PROGRAM Note
VAR
END_VAR

進料台車:
	編碼器對應實際距離: 0.025mm/p
	歸零偏移 : 22mm  > 880p
	最大行程 編碼器 108466 p 實際 2710 mm
	進料範圍 0 - 1000
	暫存範圍 1300 - 2800
	
	30HZ = 164mm/S
	 3HZ =  16mm/S
	 
進料流程:
1.將進料區的工件全部往定位住靠邊，這時候順便檢查 總和寬度 與設定的 容許誤差 做比較
2.將進料區的工件搬移到 等待區 ， 並做分料的動作。
3.將第1支搬入進料區
4.1. 台車繼續 將後續的工件 向前搬 
4.2.1 進料區做工件靠邊
4.2.2 檢測翼板高度，並向前送入雷射機
4.2.3 檢測工件寬度

5.完成進料動作


備註:
緩衝區進完最後的工件後，將再次從1開始


進料計算筆記
	臺車總長 = 1100
	
	工件待命位置= 1400
	
	第二支料分離起始位置 =  工件待命位置 + 臺車寬度 - (第一支料寬 + (第二支料寬 / 2))
	
	第二支料分離結束位置 =  工件待命位置 + 臺車寬度 - (第一支料寬 + 第二支料寬 + 材料排列間距)
	
	第三支料分離起始位置 =  工件待命位置 + 臺車寬度 - (第一支料寬 + 第二支料寬 + (第三支料寬 / 2))
	
	第三支料分離結束位置 =  工件待命位置 + 臺車寬度 - (第二支料分離結束位置 + 第三支料寬 + 材料排列間距)
	
	動作: 從最後一隻開始移動，依序往前


給料計算 筆記
	臺車總長 = 1100
	
	工件待命位置= 1400

	第一支進料移動起始位置 =  工件待命位置 + 臺車寬度 - (第一支料寬 + 材料排列間距)
	
	移動距離 = 給料位置 - 第一支進料移動起始位置
	
	移動次數 = (臺車總長 / 移動距離) ->> 取整數 ，若無小數點，直接減一

END_PROGRAM

(* stored: Version 1.1.0.1, ProductVersion 3.1.4026.13
   POU Note: Id {1b844dda-8a5b-4a3e-8835-9172b65cc59b}, SpecialFunc None *)
